(* PLC project Hardware_Configuration, BoxTurtle PicoShield_v2 2.0 *)
(* stored: creationDateTime 2025-11-21T14:00:00, modificationDateTime 2025-11-21T14:00:00 *)

CONFIGURATION BoxTurtle_Controller
  RESOURCE RaspberryPi_Pico ON PLC
    VAR_GLOBAL
      bSensor_Lane1 AT %IX0.0 : BOOL;  (* Filament Presence Sensor Lane 1 (Omron D2HW-C201H) (Pin GP16) *)
      bSensor_Lane2 AT %IX0.1 : BOOL;  (* Filament Presence Sensor Lane 2 (Omron D2HW-C201H) (Pin GP17) *)
      bSensor_Lane3 AT %IX0.2 : BOOL;  (* Filament Presence Sensor Lane 3 (Omron D2HW-C201H) (Pin GP18) *)
      bSensor_Lane4 AT %IX0.3 : BOOL;  (* Filament Presence Sensor Lane 4 (Omron D2HW-C201H) (Pin GP19) *)
      bMotor_L1_Step AT %QX0.0 : BOOL;  (* Lane 1 Stepper STEP (NEMA 14) (Pin GP2) *)
      bMotor_L1_Dir AT %QX0.1 : BOOL;  (* Lane 1 Stepper DIR (Pin GP3) *)
      bMotor_L2_Step AT %QX0.2 : BOOL;  (* Lane 2 Stepper STEP (Pin GP4) *)
      bMotor_L2_Dir AT %QX0.3 : BOOL;  (* Lane 2 Stepper DIR (Pin GP5) *)
      bMotor_L3_Step AT %QX0.4 : BOOL;  (* Lane 3 Stepper STEP (Pin GP6) *)
      bMotor_L3_Dir AT %QX0.5 : BOOL;  (* Lane 3 Stepper DIR (Pin GP7) *)
      bMotor_L4_Step AT %QX0.6 : BOOL;  (* Lane 4 Stepper STEP (Pin GP10) *)
      bMotor_L4_Dir AT %QX0.7 : BOOL;  (* Lane 4 Stepper DIR (Pin GP11) *)
      bMotor_Enable AT %QX1.0 : BOOL;  (* Shared Stepper Enable (Active Low) (Pin GP12) *)
      wServo_PWM AT %QW0 : WORD;  (* Cutter Servo PWM Duty Cycle (Pin GP20) *)
      bI2C_Status AT %IB0 : BYTE;  (* I2C Bus Status (SDA=GP14, SCL=GP15) *)
      bAux_IO1 AT %QX2.0 : BOOL;  (* Aux IO 1 / UART TX (Pin GP21) *)
      bAux_IO2 AT %QX2.1 : BOOL;  (* Aux IO 2 / UART RX (Pin GP22) *)
    END_VAR
  END_RESOURCE
END_CONFIGURATION
